Staubli VAL3: start.pgx

program start()
  local bool l_bOk
begin
  userPage()

  // if external 24V not activated, do nothing
  if hasCpuExtPowerSupply()==false
    logMsg("CPU has no external power Supply, skipped the test")
  else
    logMsg("CPU has an external power supply")
    // We can monitor main power supply failure


    l_bOk = false
    while l_bOk==false
      if dDioMainPowerOk==false
        userPageAlert("power supply failure, wait power supply ok")
        // TODO Save application data here
        // ....
        // wait for power and recover after power supply failure
        while wakeUpRobot() != 0
          delay(1)
        endWhile
        l_bOk = userPageConfirm("Press update button to complete robot restauration")
      endIf
      delay(1)
    endWhile
  endIf

end
